(* CODESYS project codesys-syslog-unit-test-history

Project tree, tasks and I/O mapping:
  Device : CODESYS Control Win V3 x64, 3S - Smart Software Solutions GmbH, version 3.5.18.0
    application Application
      libraries: Standard, 3.5.18.0 (System); co♻e - A unittest framework for CODESYS, 1.2.0.0 (www.co5e.org); Code-Syslog Interfaces, * (PowerCore Engineering); CAA File, 3.5.17.0 (CAA Technical Workgroup); CAA Types Extern, 3.5.17.0 (CAA Technical Workgroup); Net Base Services, 3.5.17.0 (3S - Smart Software Solutions GmbH); Element Collections, 3.5.17.0 (3S - Smart Software Solutions GmbH); StringUtils, 3.5.18.0 (System); Code-Syslog, 0.2.0.0 (PowerCore Engineering)
      task MainTask (cyclic, interval t#20ms, priority 1) calls PLC_PRG
      Function Blocks/
        function block UT_SyslogAlarmOnMessageHandler [ST]: T001_TripAlarm, T002_WarnAlarm, T003_RepeatAlarm, T004_RegisterDup
        function block UT_SyslogCaaUdpHandler [ST]: T002_SetupConnection, T003_ProcessQueue
        function block UT_SyslogFileHandler [ST]: AssertEquals_SyslogMsg, CleanUp, T001_FileSetup, T002_ProcessQueue, T003_DiscardWhenFull, T004_FileRemovalRecovery, T999_CleanUp
        function block UT_SyslogLogger [ST]: AssertEquals_SyslogMsg, T001_AppName, T002_Hostname, T003_ProcId, T004_HandlerRegistry, T005_Debug, T006_Info, T007_Notice, T008_Warning, T009_Error, T010_Critical, T011_Alert, T012_Emergency
        function block UT_SyslogRotatingFileHandler [ST]: CleanUp, ls_count, T001_FileSetup, T002_ShouldRollover, T003_Rotate, T004_DoRollover, T005_FullRun, T999_CleanUp
        function block UT_SyslogUdpHandler [ST]: T001_Init, T002_SetupConnection, T003_ProcessQueue
      Functions/
        function block UT_Escape_ParamValue [ST]: T001_Paramaterize
        function block UT_Make_Priority [ST]: T001_Paramaterize
        function block UT_Make_SdParam2 [ST]: T001_Parameterize
        function block UT_Make_SdParam [ST]: T001_Parameterize
        function block UT_RandomEmpherialPort [ST]: T001_Generate
        function block UT_Sanitize_Msg [ST]: T001_Paramaterize
        function block UT_Sanitize_PrintUsAscii [ST]: T001_Paramaterize
        function block UT_Sanitize_SdName [ST]: T001_Paramaterize
        function block UT_StrucDataMsg [ST]: AssertEquals_SyslogMsg, T001_Parameterize
        function block UT_UtcTimestampFromSysTimeDate [ST]: T001_Paramaterize
      Mocks/
        function block Mock_MsgPrependSpace [ST]: AsStructuredData
        function block Mock_StructuredData [ST]: AsStructuredData
        function block Mock_SyslogCaaUdpHandler [ST]: p_QueueBusy, p_uiSendPort, PubProcessQueue, PubSetupConnection, Reset
        function block Mock_SyslogFileHandler [ST]: FileSetup, FlushNow, p_DiscardOldMsgWhenQueueFull, p_FileSize, p_FullFilename, p_mxHandler, p_QueueBusy, PeekQueue, ProcessQueue, ResetQueue
        function block Mock_SyslogHandler [ST]: Dispatch, FB_Init, p_LogSeverity, Reset, Run
        function block Mock_SyslogLogger [ST]: prvTimestamp
        function block Mock_SyslogRotatingFileHandler [ST]: FileSetup, p_FileSize, p_FullFilename, p_hActiveHandle, p_mxHandler, p_QueueBusy, ProcessQueue, PubDoRollover, PubRotate, PubShouldRollover, QueueEmpty, ResetQueue
        function block Mock_SyslogUdpHandler [ST]: AdhockSend, p_QueueBusy, p_uiSendPort, PubInit, PubProcessQueue, PubSetupConnection, Reset
      program PLC_PRG [ST]
      Structs/
        data type ls_data
*)

// Device/Application/Structs/ls_data
TYPE ls_data :
STRUCT
	cFiles : INT;
	szTotalSize : CAA.SIZE;
END_STRUCT
END_TYPE

// Device/Application/PLC_PRG
PROGRAM PLC_PRG
VAR
	utSanitize_PrintUsAscii : UT_Sanitize_PrintUsAscii;
	utSanitize_SdName : UT_Sanitize_SdName;
	utSanitize_Msg : UT_Sanitize_Msg;
	utEscape_ParamValue : UT_Escape_ParamValue;
	utUtcTimestampFromSysTimeDate : UT_UtcTimestampFromSysTimeDate;
	utMake_Priority : UT_Make_Priority;
	utSyslogLogger : UT_SyslogLogger;
	utSyslogFileHandler : UT_SyslogFileHandler;
	utSyslogRotatingFileHandler : UT_SyslogRotatingFileHandler;
	utRandomEmpherialPort : UT_RandomEmpherialPort;
	utSyslogUdpHandler : UT_SyslogUdpHandler;
	utMake_SdParam : UT_Make_SdParam;
	utMake_SdParam2 : UT_Make_SdParam2;
	utStrucDataMsg : UT_StrucDataMsg;
END_VAR

coUnit.RUN_IN_SEQUENCE();

END_PROGRAM

// Device/Application/Functions/UT_Sanitize_PrintUsAscii
FUNCTION_BLOCK UT_Sanitize_PrintUsAscii EXTENDS coUnit.FB_TestSuite
VAR_INPUT
END_VAR
VAR_OUTPUT
END_VAR
VAR
END_VAR

T001_Paramaterize('LegalChars', 
                  'aValidName[don$'t-you_know]',
                  'aValidName[don$'t-you_know]');
T001_Paramaterize('StartWithIllegalChars', 
                  '$n$raValidName[don$'t-you_know]',
                  'aValidName[don$'t-you_know]');
T001_Paramaterize('EndWithIllegalChars', 
                  'aValidName[don$'t-you_know]$de$ad$be$af',
                  'aValidName[don$'t-you_know]');
T001_Paramaterize('IllegalCharsInMiddle', 
                  'aValidName[don$'t-$de$adyou$be$af_know]',
                  'aValidName[don$'t-you_know]');
T001_Paramaterize('AllLegalChars',
                  Syslog.SyslogItfs.gc_sPRINTUSASCII,
                  Syslog.SyslogItfs.gc_sPRINTUSASCII);

METHOD T001_Paramaterize : BOOL
VAR_INPUT
	sTestName : STRING(80);
	sValue : STRING(1000);
	sExpected : STRING(1000);
END_VAR
TEST(sTestName);

Syslog.Sanitize_PrintUsAscii(ADR(sValue));

AssertEquals_BOOL(TRUE, Stu.StrCmpA(ADR(sValue), ADR(sExpected)) = 0, 'sValue does not equal sExpected');

TEST_FINISHED();
END_METHOD

END_FUNCTION_BLOCK

// Device/Application/Functions/UT_Sanitize_SdName
FUNCTION_BLOCK UT_Sanitize_SdName EXTENDS coUnit.FB_TestSuite
VAR_INPUT
END_VAR
VAR_OUTPUT
END_VAR
VAR
END_VAR

T001_Paramaterize('LegalName', 
                  'eventSource',
                  'eventSource');
T001_Paramaterize('StartWithIllegalChars', 
                  '$n$reventSource',
                  'eventSource');
T001_Paramaterize('EndWithIllegalChars', 
                  'eventSource$de$ad$be$af',
                  'eventSource');
T001_Paramaterize('IllegalCharsInMiddle', 
                  'event"]= Source',
                  'eventSource');
T001_Paramaterize('AllLegalChars', 
                  '!#$$%&$'()*+,-./0123456789:;<>?@ABCDEFGHIJKLMNOPQRSTUVWXYZ[\^_`abcdefghijklmnopqrstuvwxyz{|}~',
                  '!#$$%&$'()*+,-./0123456789:;<>?@ABCDEFGHIJKLMNOPQRSTUVWXYZ[\^_`abcdefghijklmnopqrstuvwxyz{|}~');

METHOD T001_Paramaterize : BOOL
VAR_INPUT
	sTestName : STRING(80);
	sValue : STRING(255);
	sExpected : STRING(255);
END_VAR
TEST(sTestName);

Syslog.Sanitize_SdName(ADR(sValue));

AssertEquals_BOOL(TRUE, Stu.StrCmpA(ADR(sValue), ADR(sExpected)) = 0, 'sValue does not equal sExpected');

TEST_FINISHED();
END_METHOD

END_FUNCTION_BLOCK

// Device/Application/Functions/UT_Sanitize_Msg
FUNCTION_BLOCK UT_Sanitize_Msg EXTENDS coUnit.FB_TestSuite
VAR_INPUT
END_VAR
VAR_OUTPUT
END_VAR
VAR
END_VAR

T001_Paramaterize('LegalChars', 
                  '$'su root$' failed for lonvick on /dev/pts/8',
                  '$'su root$' failed for lonvick on /dev/pts/8');
T001_Paramaterize('StartWithIllegalChars', 
                  '$n$r$'su root$' failed for lonvick on /dev/pts/8',
                  '\x0a\x0d$'su root$' failed for lonvick on /dev/pts/8');
T001_Paramaterize('EndWithIllegalChars', 
                  '$'su root$' failed for lonvick on /dev/pts/8$de$ad$be$af$n$r',
                  '$'su root$' failed for lonvick on /dev/pts/8$de$ad$be$af\x0a\x0d');
T001_Paramaterize('IllegalCharsInMiddle', 
                  '$'su root$' failed $de$adfor$be$af$n$r lonvick on /dev/pts/8',
                  '$'su root$' failed $de$adfor$be$af\x0a\x0d lonvick on /dev/pts/8');
T001_Paramaterize('AllLegalChars', 
                  Syslog.SyslogItfs.gc_sPRINTUSASCII,
                  Syslog.SyslogItfs.gc_sPRINTUSASCII);

METHOD T001_Paramaterize : BOOL
VAR_INPUT
	sTestName : STRING(80);
	sValue : STRING(1000);
	sExpected : STRING(1000);
END_VAR
TEST(sTestName);

Syslog.Sanitize_Msg(ADR(sValue), sizeof(sValue));

AssertEquals_BOOL(TRUE, Stu.StrCmpA(ADR(sValue), ADR(sExpected)) = 0, 'sValue does not equal sExpected');

TEST_FINISHED();
END_METHOD

END_FUNCTION_BLOCK

// Device/Application/Functions/UT_Escape_ParamValue
FUNCTION_BLOCK UT_Escape_ParamValue EXTENDS coUnit.FB_TestSuite
VAR_INPUT
END_VAR
VAR_OUTPUT
END_VAR
VAR
END_VAR

T001_Paramaterize('LegalName', 
                  'eventSource',
                  'eventSource');
T001_Paramaterize('StartWithUnescapedChars', 
                  ']"\eventSource',
                  '\]\"\\eventSource');
T001_Paramaterize('EndWithUnescapedChars', 
                  'eventSource]"\',
                  'eventSource\]\"\\');
T001_Paramaterize('UnescapedCharsInMiddle', 
                  'event"]\Source',
                  'event\"\]\\Source');
T001_Paramaterize('MixOfEscapedAndUnescaped', 
                  'event\"\\So\ur]ce',
                  'event\"\\So\\ur\]ce');
T001_Paramaterize('AllLegalChars', 
                  '!#$$%&$'()*+,-./0123456789:;<=>?@ABCDEFGHIJKLMNOPQRSTUVWXYZ[^_`abcdefghijklmnopqrstuvwxyz{|}~',
                  '!#$$%&$'()*+,-./0123456789:;<=>?@ABCDEFGHIJKLMNOPQRSTUVWXYZ[^_`abcdefghijklmnopqrstuvwxyz{|}~');

METHOD T001_Paramaterize : BOOL
VAR_INPUT
	sTestName : STRING(80);
	sValue : STRING(255);
	sExpected : STRING(255);
END_VAR
TEST(sTestName);

Syslog.Escape_ParamValue(ADR(sValue), sizeof(sValue));

AssertEquals_BOOL(TRUE, Stu.StrCmpA(ADR(sValue), ADR(sExpected)) = 0, 'sValue does not equal sExpected');

TEST_FINISHED();
END_METHOD

END_FUNCTION_BLOCK

// Device/Application/Functions/UT_UtcTimestampFromSysTimeDate
FUNCTION_BLOCK UT_UtcTimestampFromSysTimeDate EXTENDS coUnit.FB_TestSuite
VAR_INPUT
END_VAR
VAR_OUTPUT
END_VAR
VAR
	rtsNull : Syslog.SysTimeRtc.SYSTIMEDATE;
	// 2003-10-11T22:14:15.003Z
	rtsRfcExample3 : Syslog.SysTimeRtc.SYSTIMEDATE := (wYear:=2003, wMonth:=10, wDay:=11, wHour:=22, wMinute:=14, wSecond:=15, wMilliseconds:=3);
	rtsSingleDigits : Syslog.SysTimeRtc.SYSTIMEDATE := (wYear:=2003, wMonth:=1, wDay:=1, wHour:=2, wMinute:=4, wSecond:=5, wMilliseconds:=3);
END_VAR

T001_Paramaterize('NullDate', 
                  rtsNull,
                  '0000-00-00T00:00:00.000Z');
T001_Paramaterize('RfcExample3', 
                  rtsRfcExample3,
                  '2003-10-11T22:14:15.003Z');
T001_Paramaterize('SingleDigits', 
                  rtsSingleDigits,
                  '2003-01-01T02:04:05.003Z');

METHOD T001_Paramaterize : BOOL
VAR_INPUT
	sTestName : STRING(80);
	rts : Syslog.SysTimeRtc.SYSTIMEDATE;
	sExpected : STRING(255);
END_VAR
VAR
	sTimestamp : Syslog.SyslogItfs.TIMESTAMP;
END_VAR
TEST(sTestName);

sTimestamp := Syslog.UtcTimestampFromSystimeDate(rts);

AssertEquals_STRING(sExpected, sTimestamp, 'Timestamps do not match');

TEST_FINISHED();
END_METHOD

END_FUNCTION_BLOCK

// Device/Application/Functions/UT_Make_Priority
FUNCTION_BLOCK UT_Make_Priority EXTENDS coUnit.FB_TestSuite
VAR_INPUT
END_VAR
VAR_OUTPUT
END_VAR
VAR
END_VAR

T001_Paramaterize('Kern emerg', Syslog.SyslogItfs.SyslogSeverity.EMERGENCY, Syslog.SyslogItfs.SyslogFacility.KERN, '<0>');
T001_Paramaterize('user alert', Syslog.SyslogItfs.SyslogSeverity.ALERT, Syslog.SyslogItfs.SyslogFacility.USER, '<9>');
T001_Paramaterize('local notice', Syslog.SyslogItfs.SyslogSeverity.NOTICE, Syslog.SyslogItfs.SyslogFacility.LOCAL4, '<165>');

METHOD T001_Paramaterize : BOOL
VAR_INPUT
	sTestName : STRING(255);
	sev : Syslog.SyslogItfs.SyslogSeverity;
	fac : Syslog.SyslogItfs.SyslogFacility;
	sExpected : STRING(10);
END_VAR
VAR
	pri : Syslog.SyslogItfs.PRI;
END_VAR
TEST(sTestName);

pri := Syslog.Make_Priority(sev, fac);

AssertEquals_STRING(pri, sExpected, 'PRI does not equal sExpected');

TEST_FINISHED();
END_METHOD

END_FUNCTION_BLOCK

// Device/Application/Function Blocks/UT_SyslogLogger
FUNCTION_BLOCK UT_SyslogLogger EXTENDS coUnit.FB_TestSuite
VAR_INPUT
END_VAR
VAR_OUTPUT
END_VAR
VAR
	handler : Mock_SyslogHandler(severity:=SyslogItfs.SyslogSeverity.DEBUG);
	itfHandler : SyslogItfs.ISyslogHandler := handler;
	// local4 = 20 to make manual pri easier to calculate. 20*8 = 160
	logger : Mock_SyslogLogger(hostname:='codesyslog.example.com', appName:='UnitTest', procId:='PLC_PRG', facility:=SyslogItfs.SyslogFacility.LOCAL4, handler:=itfHandler);
END_VAR

T001_AppName('T001_AppName:EmptyAppName', '', SyslogItfs.gc_sNILVALUE);
T001_AppName('T001_AppName:InvalidCharsRemoved', '$nUnit Test', 'UnitTest');

T002_Hostname('T002_Hostname:EmptyHostname', '$n $r', SyslogItfs.gc_sNILVALUE);
T002_Hostname('T002_Hostname:InvalidCharsRemoved', 'invalid hostname', 'invalidhostname');
T002_Hostname('T002_Hostname:IPAddress', '192.168.0.1', '192.168.0.1');
T002_Hostname('T002_Hostname:FQDN', 'codesyslog.example.com', 'codesyslog.example.com');

T003_ProcId('T003_ProcId:EmptyProcId', '', SyslogItfs.gc_sNILVALUE);
T003_ProcId('T003_ProcId:InvalidCharsRemoved', '$de$ad$be$efPLC_PRG', 'PLC_PRG');

T004_HandlerRegistry();
T005_Debug();
T006_Info();
T007_Notice();
T008_Warning();
T009_Error();
T010_Critical();
T011_Alert();
T012_Emergency();

METHOD AssertEquals_SyslogMsg
VAR_INPUT
	actual : POINTER TO SyslogItfs.SYSLOG_MSG;
	expected : POINTER TO SyslogItfs.SYSLOG_MSG;
END_VAR
VAR
	ix : UINT;
	pa : POINTER TO ARRAY [0..SyslogItfs.gc_szSyslogMsg-1] OF BYTE := actual;
	pe : POINTER TO ARRAY [0..SyslogItfs.gc_szSyslogMsg-1] OF BYTE := expected;
	xDifferent : BOOL;
END_VAR
FOR ix := 0 TO SyslogItfs.gc_szSyslogMsg-1 BY 1 DO
	IF pa^[ix] <> 0 AND pe^[ix] <> 0 THEN
		IF pa^[ix] <> pe^[ix] THEN
			xDifferent := TRUE;
			EXIT;
		END_IF
	ELSIF pa^[ix] = 0 AND pe^[ix] = 0 THEN
		EXIT;
	ELSE
		xDifferent := TRUE;
		EXIT;
	END_IF
END_FOR

AssertFalse(xDifferent, concat('SYSLOG_MSG found to differ at character: ', UINT_TO_STRING(ix)));
END_METHOD

METHOD T001_AppName
VAR_INPUT
	sTestName : STRING(255);
	sAppName : SyslogItfs.APP_NAME;
	sExpected : SyslogItfs.APP_NAME;
END_VAR
VAR
	sResult : SyslogItfs.APP_NAME;
END_VAR
IF TEST_ORDERED(sTestName) THEN

	logger.SetAppName(sAppName);
	sResult := logger.GetAppName();
	
	AssertEquals_STRING(sExpected, sResult, 'Unexpected AppName');
	
	TEST_FINISHED();
END_IF
END_METHOD

METHOD T002_Hostname
VAR_INPUT
	sTestName : STRING(255);
	sValue : SyslogItfs.HOSTNAME;
	sExpected : SyslogItfs.HOSTNAME;
END_VAR
VAR
	sResult : SyslogItfs.HOSTNAME;
END_VAR
IF TEST_ORDERED(sTestName) THEN

	logger.SetHostname(sValue);
	sResult := logger.GetHostname();
	
	AssertEquals_STRING(sExpected, sResult, 'Unexpected Hostname');
	
	TEST_FINISHED();
END_IF
END_METHOD

METHOD T003_ProcId
VAR_INPUT
	sTestName : STRING(255);
	sValue : SyslogItfs.PROC_ID;
	sExpected : SyslogItfs.PROC_ID;
END_VAR
VAR
	sResult : SyslogItfs.PROC_ID;
END_VAR
IF TEST_ORDERED(sTestName) THEN

	logger.SetProcId(sValue);
	sResult := logger.GetProcId();
	
	AssertEquals_STRING(sExpected, sResult, 'Unexpected Proc ID');
	
	TEST_FINISHED();
END_IF
END_METHOD

METHOD T004_HandlerRegistry
VAR_INPUT
END_VAR
VAR
	xResult : BOOL;
END_VAR
IF TEST_ORDERED('T004_HandlerRegistry') THEN

	xResult := logger.RegisterHandler(itfHandler);
	AssertFalse(xResult, 'Handle registered twice!');
	
	xResult := logger.UnregisterHandler(itfHandler);
	AssertTrue(xResult, 'Handle failed to unregistered');
	
	xResult := logger.RegisterHandler(itfHandler);
	AssertTrue(xResult, 'Handle failed to registered');
	
	TEST_FINISHED();
END_IF
END_METHOD

METHOD T005_Debug
VAR_INPUT
END_VAR
VAR
	expected : SyslogItfs.SYSLOG_MSG;
END_VAR
IF TEST_ORDERED('T005_Debug') THEN

	logger.Debug('DEBUG', 'lorum ipsum');
	expected := '<167>1 2021-11-22T23:40:05.003Z codesyslog.example.com UnitTest PLC_PRG DEBUG lorum ipsum';
	AssertEquals_SyslogMsg(ADR(handler.lastMessage), ADR(expected));
	
	handler.Reset();
	handler.p_LogSeverity := SyslogItfs.SyslogSeverity.INFORMATION;
	
	logger.Debug('DEBUG', 'lorum ipsum');
	expected := '';
	AssertEquals_SyslogMsg(ADR(handler.lastMessage), ADR(expected));
	
	
	TEST_FINISHED();
END_IF
END_METHOD

METHOD T006_Info
VAR_INPUT
END_VAR
VAR
	expected : SyslogItfs.SYSLOG_MSG;
END_VAR
IF TEST_ORDERED('T006_Info') THEN

	logger.Information('INFO', 'lorum ipsum');
	expected := '<166>1 2021-11-22T23:40:05.003Z codesyslog.example.com UnitTest PLC_PRG INFO lorum ipsum';
	AssertEquals_SyslogMsg(ADR(handler.lastMessage), ADR(expected));
	
	handler.Reset();
	handler.p_LogSeverity := SyslogItfs.SyslogSeverity.NOTICE;
	
	logger.Information('INFO', 'lorum ipsum');
	expected := '';
	AssertEquals_SyslogMsg(ADR(handler.lastMessage), ADR(expected));
	
	
	TEST_FINISHED();
END_IF
END_METHOD

METHOD T007_Notice
VAR_INPUT
END_VAR
VAR
	expected : SyslogItfs.SYSLOG_MSG;
END_VAR
IF TEST_ORDERED('T007_Notice') THEN

	logger.Notice('NOTICE', 'lorum ipsum');
	expected := '<165>1 2021-11-22T23:40:05.003Z codesyslog.example.com UnitTest PLC_PRG NOTICE lorum ipsum';
	AssertEquals_SyslogMsg(ADR(handler.lastMessage), ADR(expected));
	
	handler.Reset();
	handler.p_LogSeverity := SyslogItfs.SyslogSeverity.WARNING;
	
	logger.Notice('NOTICE', 'lorum ipsum');
	expected := '';
	AssertEquals_SyslogMsg(ADR(handler.lastMessage), ADR(expected));
	
	
	TEST_FINISHED();
END_IF
END_METHOD

METHOD T008_Warning
VAR_INPUT
END_VAR
VAR
	expected : SyslogItfs.SYSLOG_MSG;
END_VAR
IF TEST_ORDERED('T008_Warning') THEN

	logger.Warning('WARN', 'lorum ipsum');
	expected := '<164>1 2021-11-22T23:40:05.003Z codesyslog.example.com UnitTest PLC_PRG WARN lorum ipsum';
	AssertEquals_SyslogMsg(ADR(handler.lastMessage), ADR(expected));
	
	handler.Reset();
	handler.p_LogSeverity := SyslogItfs.SyslogSeverity.ERROR;
	
	logger.Warning('WARN', 'lorum ipsum');
	expected := '';
	AssertEquals_SyslogMsg(ADR(handler.lastMessage), ADR(expected));
	
	
	TEST_FINISHED();
END_IF
END_METHOD

METHOD T009_Error
VAR_INPUT
END_VAR
VAR
	expected : SyslogItfs.SYSLOG_MSG;
END_VAR
IF TEST_ORDERED('T009_Error') THEN

	logger.Error('ERROR', 'lorum ipsum');
	expected := '<163>1 2021-11-22T23:40:05.003Z codesyslog.example.com UnitTest PLC_PRG ERROR lorum ipsum';
	AssertEquals_SyslogMsg(ADR(handler.lastMessage), ADR(expected));
	
	handler.Reset();
	handler.p_LogSeverity := SyslogItfs.SyslogSeverity.CRITICAL;
	
	logger.Error('ERROR', 'lorum ipsum');
	expected := '';
	AssertEquals_SyslogMsg(ADR(handler.lastMessage), ADR(expected));
	
	
	TEST_FINISHED();
END_IF
END_METHOD

METHOD T010_Critical
VAR_INPUT
END_VAR
VAR
	expected : SyslogItfs.SYSLOG_MSG;
END_VAR
IF TEST_ORDERED('T010_Critical') THEN

	logger.Critical('CRITICAL', 'lorum ipsum');
	expected := '<162>1 2021-11-22T23:40:05.003Z codesyslog.example.com UnitTest PLC_PRG CRITICAL lorum ipsum';
	AssertEquals_SyslogMsg(ADR(handler.lastMessage), ADR(expected));
	
	handler.Reset();
	handler.p_LogSeverity := SyslogItfs.SyslogSeverity.ALERT;
	
	logger.Critical('CRITICAL', 'lorum ipsum');
	expected := '';
	AssertEquals_SyslogMsg(ADR(handler.lastMessage), ADR(expected));
	
	
	TEST_FINISHED();
END_IF
END_METHOD

METHOD T011_Alert
VAR_INPUT
END_VAR
VAR
	expected : SyslogItfs.SYSLOG_MSG;
END_VAR
IF TEST_ORDERED('T011_Alert') THEN

	logger.Alert('ALERT', 'lorum ipsum');
	expected := '<161>1 2021-11-22T23:40:05.003Z codesyslog.example.com UnitTest PLC_PRG ALERT lorum ipsum';
	AssertEquals_SyslogMsg(ADR(handler.lastMessage), ADR(expected));
	
	handler.Reset();
	handler.p_LogSeverity := SyslogItfs.SyslogSeverity.EMERGENCY;
	
	logger.Alert('ALERT', 'lorum ipsum');
	expected := '';
	AssertEquals_SyslogMsg(ADR(handler.lastMessage), ADR(expected));
	
	
	TEST_FINISHED();
	END_IF
END_METHOD

METHOD T012_Emergency
VAR_INPUT
END_VAR
VAR
	expected : SyslogItfs.SYSLOG_MSG;
END_VAR
IF TEST_ORDERED('T012_Emergency') THEN

	logger.Emergency('EMERGENCY', 'lorum ipsum');
	expected := '<160>1 2021-11-22T23:40:05.003Z codesyslog.example.com UnitTest PLC_PRG EMERGENCY lorum ipsum';
	AssertEquals_SyslogMsg(ADR(handler.lastMessage), ADR(expected));
	
	handler.Reset();
	handler.p_LogSeverity := SyslogItfs.SyslogSeverity.DEBUG;
	
	logger.Emergency('EMERGENCY', 'lorum ipsum debug');
	expected := '<160>1 2021-11-22T23:40:05.003Z codesyslog.example.com UnitTest PLC_PRG EMERGENCY lorum ipsum debug';
	AssertEquals_SyslogMsg(ADR(handler.lastMessage), ADR(expected));
	
	
	TEST_FINISHED();
END_IF
END_METHOD

END_FUNCTION_BLOCK

// Device/Application/Mocks/Mock_SyslogHandler
/// This syslog handler doesn't only stores the last value dispatched
FUNCTION_BLOCK Mock_SyslogHandler IMPLEMENTS SyslogItfs.ISyslogHandler
VAR_INPUT
END_VAR
VAR_OUTPUT
	lastMessage : SyslogItfs.SYSLOG_MSG;
END_VAR
VAR
	_severity : SyslogItfs.SyslogSeverity;
END_VAR

METHOD Dispatch : BOOL
VAR_INPUT
	syslogMsg	: SyslogItfs.SYSLOG_MSG;
END_VAR
THIS^.lastMessage := syslogMsg;
END_METHOD

//FB_Init is always available implicitly and it is used primarily for initialization.
//The return value is not evaluated. For a specific influence, you can also declare the
//methods explicitly and provide additional code there with the standard initialization
//code. You can evaluate the return value.
METHOD FB_Init: BOOL
VAR_INPUT
    bInitRetains: BOOL; // TRUE: the retain variables are initialized (reset warm / reset cold)
    bInCopyCode: BOOL;  // TRUE: the instance will be copied to the copy code afterward (online change)   
	severity : SyslogItfs.SyslogSeverity;
END_VAR
THIS^._severity := severity;
END_METHOD

{attribute 'monitoring' := 'call'}
PROPERTY p_LogSeverity : SyslogItfs.SyslogSeverity
GET
p_LogSeverity := this^._severity;
END_GET
SET
this^._severity := p_LogSeverity;
END_SET
END_PROPERTY

METHOD Reset : BOOL
VAR_INPUT
END_VAR
lastMessage := '';
END_METHOD

(* Run the handler base code*)
METHOD Run : BOOL
END_METHOD

END_FUNCTION_BLOCK

// Device/Application/Mocks/Mock_SyslogLogger
FUNCTION_BLOCK Mock_SyslogLogger EXTENDS Syslog.SyslogLogger
VAR_INPUT
END_VAR
VAR_OUTPUT
END_VAR
VAR
END_VAR

/// prvTimestamp exists so we can override the timestamp for testing
METHOD PROTECTED prvTimestamp : Syslog.SyslogItfs.TIMESTAMP
VAR_INPUT
END_VAR
VAR
	// 2021-11-22T23:40:05.003Z
	rts : Syslog.SysTimeRtc.SYSTIMEDATE := (wYear:=2021, wMonth:=11, wDay:=22, wHour:=23, wMinute:=40, wSecond:=5, wMilliseconds:=3);
END_VAR
prvTimestamp := Syslog.UtcTimestampFromSystimeDate(rts);
END_METHOD

END_FUNCTION_BLOCK

// Device/Application/Function Blocks/UT_SyslogFileHandler
FUNCTION_BLOCK UT_SyslogFileHandler EXTENDS coUnit.FB_TestSuite
VAR_INPUT
END_VAR
VAR_OUTPUT
END_VAR
VAR
	handler : Mock_SyslogFileHandler;
END_VAR

T001_FileSetup();
T002_ProcessQueue();
T003_DiscardWhenFull();
T004_FileRemovalRecovery();


// Final cleanup
T999_CleanUp();

METHOD AssertEquals_SyslogMsg
VAR_INPUT
	actual : POINTER TO SyslogItfs.SYSLOG_MSG;
	expected : POINTER TO SyslogItfs.SYSLOG_MSG;
END_VAR
VAR
	ix : UINT;
	pa : POINTER TO ARRAY [0..SyslogItfs.gc_szSyslogMsg-1] OF BYTE := actual;
	pe : POINTER TO ARRAY [0..SyslogItfs.gc_szSyslogMsg-1] OF BYTE := expected;
	xDifferent : BOOL;
END_VAR
FOR ix := 0 TO SyslogItfs.gc_szSyslogMsg-1 BY 1 DO
	IF pa^[ix] <> 0 AND pe^[ix] <> 0 THEN
		IF pa^[ix] <> pe^[ix] THEN
			xDifferent := TRUE;
			EXIT;
		END_IF
	ELSIF pa^[ix] = 0 AND pe^[ix] = 0 THEN
		EXIT;
	ELSE
		xDifferent := TRUE;
		EXIT;
	END_IF
END_FOR

AssertFalse(xDifferent, concat('SYSLOG_MSG found to differ at character: ', UINT_TO_STRING(ix)));
END_METHOD

METHOD CleanUp : BOOL;
VAR_INPUT
END_VAR
VAR_INST
	rmdir : FILE.DirRemove;
END_VAR
rmdir(xExecute:=TRUE, sDirName:='csyslog/', xRecursive:=TRUE);
IF rmdir.xDone OR rmdir.xError THEN
	CleanUp := TRUE;
	rmdir(xExecute:=FALSE);
END_IF
END_METHOD

METHOD T001_FileSetup
VAR_INPUT
END_VAR
VAR_INST
	tmr : TON := (PT:=T#5S);
	mxFileSetup : UINT;
	getSize : FILE.GetSize;
END_VAR
IF TEST_ORDERED('T001_FileSetup') THEN
	tmr(IN:=TRUE);
	CASE mxFileSetup OF
		0: // Run file setup
			IF handler.FileSetup() OR tmr.Q OR handler.xError THEN
				mxFileSetup := 10;
			END_IF
		10: // Simple Asserts
			AssertFalse(handler.xError, 'Error after file setup');
			AssertFalse(tmr.Q, 'FileSetup timed out');
			mxFileSetup := 20;
		20: // check filesystem
			getSize(xExecute:=TRUE, sFileName:=handler.p_FullFilename);
			IF getSize.xDone OR getSize.xError THEN
				AssertFalse(getSize.xError, concat('An error occured getting file size. Error: ', TO_STRING(getSize.eError)));
				AssertFalse(getSize.xError, concat('Error on file: ', TO_STRING(handler.p_FullFilename)));
				getSize(xExecute:=FALSE);
				mxFileSetup := 30;
			END_IF
		ELSE
			TEST_FINISHED();
	END_CASE
	
	
END_IF
END_METHOD

METHOD T002_ProcessQueue
VAR_INPUT
END_VAR
VAR_INST
	mxT : UINT;
	tmr : TON := (PT:=T#5S);
	fileSize : FILE.GetSize;
END_VAR
IF TEST_ORDERED('T002_ProcessQueue') THEN
	CASE mxT OF
		0: // setup
			handler.Dispatch('hello, world');
			handler.Dispatch('<167>1 2021-11-22T23:40:05.003Z codesyslog.example.com UnitTest PLC_PRG DEBUG lorum ipsum');
			mxT := 10;
		10: // run queue process for 5 seconds
			tmr(IN:=TRUE);
			handler.ProcessQueue();
			IF tmr.Q OR NOT handler.p_QueueBusy THEN
				AssertFalse(tmr.Q, 'ProcessQueue timeout');
				tmr(IN:=FALSE);
				mxT := 20;
			END_IF
		20: // get fileSize
			fileSize(xExecute:=TRUE, sFileName:=handler.p_FullFilename);
			IF fileSize.xDone OR fileSize.xError THEN
				AssertFalse(fileSize.xError, 'Error getting file size');
				AssertEquals_UDINT(handler.p_FileSize, __UXINT_TO_UDINT(fileSize.szSize), 'calculated file size and actual file size do not match');
				fileSize(xExecute:=FALSE); 
				mxT := 30;
			END_IF
		30: // other asserts
			AssertFalse(handler.xError, 'Error during queue processing');
			mxT := 40;
		ELSE
			TEST_FINISHED();
	END_CASE
END_IF
END_METHOD

METHOD T003_DiscardWhenFull
VAR_INPUT
END_VAR
VAR_INST
	mxT : UINT;
	ix : UINT;
	sHead : SyslogItfs.SYSLOG_MSG;
	sExpected : STRING(10) := '21';
END_VAR
IF TEST_ORDERED('T003_DiscardWhenFull') THEN
	CASE mxT OF
		0: // init
			handler.p_DiscardOldMsgWhenQueueFull := TRUE;
			FOR ix := 0 TO 1020 BY 1 DO
				handler.Dispatch(UINT_TO_STRING(ix));
			END_FOR
			mxT := 10;
		10: // check for overrun
			sHead := handler.PeekQueue();
			AssertEquals_STRING(sExpected, sHead, 'Queue head unexpected value');
			handler.ResetQueue();
			handler.p_DiscardOldMsgWhenQueueFull := FALSE;
			mxT := 20;
		ELSE
			TEST_FINISHED();
	END_CASE
END_IF
END_METHOD

METHOD T004_FileRemovalRecovery
VAR_INPUT
END_VAR
VAR_INST
	mxT : UINT;
	tmr : TON := (PT:=T#10s);
END_VAR
IF TEST_ORDERED('T004_FileRemovalRecovery') THEN
	CASE mxT OF
		0: // setup
			// run until in process queue
			handler.Run();
			IF handler.p_mxHandler = 10 THEN
				// remove directory and file
				IF CleanUp() THEN
					mxT := 10;
				END_IF
			END_IF
		10: // dispatch a message
			handler.Dispatch('write to missing file');
			mxT := 20;
		20: // run until back in init mode
			handler.Run();
			tmr(IN:=TRUE);
			IF handler.p_mxHandler = 0 OR tmr.Q THEN
				AssertFalse(tmr.Q, 'handler.Run() until timeout mxT=20');
				AssertFalse(handler.xError, 'handler.xError mxT=20');
				tmr(IN:=FALSE);
				mxT := 30;
			END_IF
		30: // run until idle (should never have stopped being busy during reset)
			handler.Run();
			tmr(IN:=TRUE);
			IF (handler.p_mxHandler = 10 AND NOT handler.p_QueueBusy) OR tmr.Q THEN
				AssertFalse(tmr.Q, 'handler.Run() until timeout mxT=30');
				AssertFalse(handler.xError, 'handler.xError mxT=30');
				mxT := 40;
			END_IF
		ELSE
			TEST_FINISHED();
	END_CASE
END_IF
END_METHOD

METHOD T999_CleanUp
VAR_INPUT
END_VAR
IF TEST_ORDERED('T999_CleanUp') THEN
	IF CleanUp() THEN
		AssertTrue(TRUE, 'cleaned up');
		TEST_FINISHED();
	END_IF
END_IF
END_METHOD

END_FUNCTION_BLOCK

// Device/Application/Mocks/Mock_SyslogFileHandler
FUNCTION_BLOCK Mock_SyslogFileHandler EXTENDS Syslog.SyslogFileHandler
VAR_INPUT
END_VAR
VAR_OUTPUT
END_VAR
VAR
END_VAR

METHOD FileSetup : BOOL
VAR_INPUT
END_VAR
FileSetup := prvFileSetup();
END_METHOD

METHOD FlushNow : BOOL
VAR_INPUT
END_VAR
FlushNow := THIS^.prvFlush();
END_METHOD

PROPERTY p_DiscardOldMsgWhenQueueFull : BOOL
GET
p_DiscardOldMsgWhenQueueFull := THIS^.xDiscardOldMsgWhenQueueFull;
END_GET
SET
THIS^.xDiscardOldMsgWhenQueueFull := p_DiscardOldMsgWhenQueueFull;
END_SET
END_PROPERTY

{attribute 'monitoring' := 'call'}
PROPERTY p_FileSize : UDINT
GET
p_FileSize := THIS^.szFilesize;
END_GET
END_PROPERTY

{attribute 'monitoring' := 'call'}
PROPERTY p_FullFilename : CAA.FILENAME
GET
p_FullFilename := THIS^.sFullFilename;
END_GET
END_PROPERTY

PROPERTY p_mxHandler : UINT
GET
p_mxHandler := mxHandler;
END_GET
END_PROPERTY

PROPERTY p_QueueBusy : BOOL
GET
p_QueueBusy := xQueueBusy;
END_GET
END_PROPERTY

METHOD PeekQueue : SyslogItfs.SYSLOG_MSG
VAR_INPUT
END_VAR
queue.Peek(itfElement => THIS^.itfElement);
IF __QUERYINTERFACE(itfElement, itfSyslogMsgElement) THEN
	PeekQueue := itfSyslogMsgElement.SyslogMsgValue;
END_IF
END_METHOD

METHOD ProcessQueue : BOOL
VAR_INPUT
END_VAR
ProcessQueue := prvProcessQueue();
END_METHOD

METHOD ResetQueue : BOOL
VAR_INPUT
END_VAR
this^.queue.RemoveAllElements();
END_METHOD

END_FUNCTION_BLOCK

// Device/Application/Function Blocks/UT_SyslogRotatingFileHandler
FUNCTION_BLOCK UT_SyslogRotatingFileHandler EXTENDS coUnit.FB_TestSuite
VAR_INPUT
END_VAR
VAR_OUTPUT
END_VAR
VAR
	handler : Mock_SyslogRotatingFileHandler := (szMaxFilesize:=1024, uiBackupCount:=3);
END_VAR

T001_FileSetup();
T002_ShouldRollover();
T003_Rotate();
T004_DoRollover();
T005_FullRun();

//T999_CleanUp();

METHOD CleanUp : BOOL;
VAR_INPUT
END_VAR
VAR_INST
	rmdir : FILE.DirRemove;
END_VAR
rmdir(xExecute:=TRUE, sDirName:='csyslog/', xRecursive:=TRUE);
IF rmdir.xDone OR rmdir.xError THEN
	CleanUp := TRUE;
	rmdir(xExecute:=FALSE);
END_IF
END_METHOD

METHOD ls_count : ls_data
VAR_INPUT
END_VAR
VAR_INST
	mxT : UINT;
	hDir : CAA.HANDLE;
	dopen : FILE.DirOpen;
	dclose : FILE.DirClose;
	dls : FILE.DirList;
	lsd : ls_data;
END_VAR
ls_count.cFiles := -1;
CASE mxT OF
	0: // open dir
		lsd.cFiles := 0;
		lsd.szTotalSize := 0;
		dopen(xExecute:=TRUE, sDirName:='csyslog/');
		IF dopen.xDone OR dopen.xError THEN
			AssertFalse(dopen.xError, 'Error opening dir');
			hDir := dopen.hDir;
			dopen(xExecute:=FALSE);
			mxT := 20;
		END_IF
	20: // list and count files
		dls(xExecute:=TRUE, hDir:=hDir);
		IF dls.xDone OR dls.xError THEN
			IF NOT dls.xError THEN
				IF dls.deDirEntry.sEntry <> '.' AND dls.deDirEntry.sEntry <> '..' THEN
					lsd.cFiles := lsd.cFiles + 1;
					lsd.szTotalSize := lsd.szTotalSize + dls.deDirEntry.szSize;
				END_IF
			ELSE
				mxT := 30;
			END_IF
			dls(xExecute:=FALSE);
		END_IF
	30: // close dir
		dclose(xExecute:=TRUE, hDir:=hDir);
		IF dclose.xDone OR dclose.xError THEN
			hDir := CAA.gc_hINVALID;
			dclose(xExecute:=FALSE);
			mxT := 0;
			ls_count := lsd;
		END_IF
END_CASE
END_METHOD

METHOD T001_FileSetup
VAR_INPUT
END_VAR
VAR_INST
	tmr : TON := (PT:=T#5S);
	mxFileSetup : UINT;
	getSize : FILE.GetSize;
END_VAR
IF TEST_ORDERED('T001_FileSetup') THEN
	tmr(IN:=TRUE);
	CASE mxFileSetup OF
		0: // Run file setup
			IF handler.FileSetup() OR tmr.Q OR handler.xError THEN
				mxFileSetup := 10;
			END_IF
		10: // Simple Asserts
			AssertFalse(handler.xError, 'Error after file setup');
			AssertFalse(tmr.Q, 'FileSetup timed out');
			mxFileSetup := 20;
		20: // check filesystem
			getSize(xExecute:=TRUE, sFileName:=handler.p_FullFilename);
			IF getSize.xDone OR getSize.xError THEN
				AssertFalse(getSize.xError, concat('An error occured getting file size. Error: ', TO_STRING(getSize.eError)));
				AssertFalse(getSize.xError, concat('Error on file: ', TO_STRING(handler.p_FullFilename)));
				getSize(xExecute:=FALSE);
				mxFileSetup := 30;
			END_IF
		ELSE
			TEST_FINISHED();
	END_CASE
	
	
END_IF
END_METHOD

METHOD T002_ShouldRollover
VAR_INPUT
END_VAR
VAR
	xResult : BOOL;
END_VAR
IF TEST_ORDERED('T002_ShouldRollover') THEN
	handler.p_FileSize := UDINT#1024;
	xResult := handler.PubShouldRollover();
	AssertFalse(xResult, 'completely full, but no message in queue');
	
	// add a message
	handler.Dispatch('hello, world'); // 12 bytes + $n = 13 bytes
	
	handler.p_FileSize := UDINT#1024 - 13;
	xResult := handler.PubShouldRollover();
	AssertFalse(xResult, 'should completely fill, but not rollover yet');
	
	handler.p_FileSize := UDINT#1024 - 12;
	xResult := handler.PubShouldRollover();
	AssertTrue(xResult, 'should rollover');
	
	handler.p_FileSize := 0;
	xResult := handler.PubShouldRollover();
	AssertFalse(xResult, 'should not rollover at 0');
	
	// reset handler
	handler.p_FileSize := 0;
	handler.ResetQueue();
	
	TEST_FINISHED();
END_IF
END_METHOD

METHOD T003_Rotate
VAR_INPUT
END_VAR
VAR_INST
	mxT : UINT;
	hHandle : CAA.HANDLE;
	sDest : CAA.FILENAME;
	fileSize : FILE.GetSize;
END_VAR
IF TEST_ORDERED('T003_Rotate') THEN
	CASE mxT OF
		0: // init
			hHandle := handler.p_hActiveHandle;
			sDest := concat(handler.p_FullFilename, '.1');
			mxT := 10;
		10: // rotate
			IF handler.PubRotate(handler.p_FullFilename, sDest) THEN
				mxT := 20;
			END_IF
		20: // get size
			fileSize(xExecute:=TRUE, sFileName:=sDest);
			IF fileSize.xError OR fileSize.xDone THEN
				AssertFalse(filesize.xError, 'sDest file should exist, but does not');
				fileSize(xExecute:=FALSE);
				mxT := 30;
			END_IF
		30: // check handle
			// we aren't guarenteed a new handle pointer value even if we close and open a file.
			//AssertFalse(CAA.HANDLE_TO_DWORD(hHandle) = CAA.HANDLE_TO_DWORD(handler.p_hActiveHandle), 'should have a new file handle');
			AssertFalse(CAA.gc_hINVALID = CAA.HANDLE_TO_DWORD(handler.p_hActiveHandle), 'should be a valid handle');
			mxT := 40;
		ELSE
			TEST_FINISHED();
	END_CASE
END_IF
END_METHOD

METHOD T004_DoRollover
VAR_INPUT
END_VAR
VAR_INST
	mxT: UINT;
	lsd : ls_data;
END_VAR
IF TEST_ORDERED('T004_DoRollover') THEN
	CASE mxT OF
		0: // Do the roll over
			IF handler.PubDoRollover() THEN
				mxT := 10;
			END_IF
		10: // count files
			lsd := ls_count();
			IF lsd.cFiles >= 0 THEN
				mxT := 40;
			END_IF
		40: // asserts
			AssertEquals_INT(3, lsd.cFiles, 'unexpected number of files after rollover');
			mxT := 50;
		ELSE
			TEST_FINISHED();
	END_CASE
END_IF
END_METHOD

METHOD T005_FullRun
VAR_INPUT
END_VAR
VAR_INST
	mxT : UINT;
	ix : UINT;
	msg : SyslogItfs.SYSLOG_MSG := ' ';
	sRow : STRING(1) := '1';
	tickStart : CAA.TICK;
	tickEnd : CAA.TICK;
	tickDiff : CAA.TICK;
	lsd : ls_data;
	szExpected : CAA.SIZE := 3328; // 13 * 256
END_VAR
IF TEST_ORDERED('T005_FullRun') THEN
	CASE mxT OF 
		0: // fill queue with enough data for 4 DoRollover
			FOR ix := 0 TO 12 BY 1 DO
				sRow := UINT_TO_STRING(ix);
				Stu.StrPadLeftA(UINT_TO_BYTE(ix) + SyslogItfs.gc_byZERO_DIGIT, ADR(sRow), ADR(msg), 255);
				handler.Dispatch(msg);
			END_FOR
			mxT := 10;
			tickStart := FILE.TICKS.GetTick(TRUE);
		10: // run until done
			handler.Run();
			IF handler.QueueEmpty() AND NOT handler.p_QueueBusy THEN
				handler.p_FlushNow := TRUE;
				mxT := 15;
				tickEnd := FILE.TICKS.GetTick(TRUE);
				tickDiff := tickEnd - tickStart;
			END_IF
		15: // run until flush done
			handler.Run();
			IF NOT handler.p_FlushNow THEN
				mxT := 20;
			END_IF
		20: // number of files
			lsd := ls_count();
			IF lsd.cFiles >= 0 THEN
				mxT := 30;
			END_IF
		30: // asserts
			AssertEquals_INT(4, lsd.cFiles, 'Unexpected number of files');
			AssertEquals(szExpected, lsd.szTotalSize, 'Unexpected file size total');
			mxT := 40;
		ELSE
			TEST_FINISHED();
	END_CASE
END_IF
END_METHOD

METHOD T999_CleanUp
VAR_INPUT
END_VAR
IF TEST_ORDERED('T999_CleanUp') THEN
	IF CleanUp() THEN
		AssertTrue(TRUE, 'cleaned up');
		TEST_FINISHED();
	END_IF
END_IF
END_METHOD

END_FUNCTION_BLOCK

// Device/Application/Mocks/Mock_SyslogRotatingFileHandler
FUNCTION_BLOCK Mock_SyslogRotatingFileHandler EXTENDS Syslog.SyslogRotatingFileHandler
VAR_INPUT
END_VAR
VAR_OUTPUT
END_VAR
VAR
END_VAR

METHOD FileSetup : BOOL
VAR_INPUT
END_VAR
FileSetup := prvFileSetup();
END_METHOD

{attribute 'monitoring' := 'call'}
PROPERTY p_FileSize : UDINT
GET
p_FileSize := THIS^.szFilesize;
END_GET
SET
THIS^.szFilesize := p_FileSize;
END_SET
END_PROPERTY

{attribute 'monitoring' := 'call'}
PROPERTY p_FullFilename : CAA.FILENAME
GET
p_FullFilename := THIS^.sFullFilename;
END_GET
END_PROPERTY

PROPERTY p_hActiveHandle : CAA.HANDLE
GET
p_hActiveHandle := THIS^.hActiveFile;
END_GET
END_PROPERTY

PROPERTY p_mxHandler : UINT
GET
p_mxHandler := mxHandler;
END_GET
END_PROPERTY

PROPERTY p_QueueBusy : BOOL
GET
p_QueueBusy := xQueueBusy;
END_GET
END_PROPERTY

METHOD ProcessQueue : BOOL
VAR_INPUT
END_VAR
ProcessQueue := prvProcessQueue();
END_METHOD

METHOD PubDoRollover : BOOL
VAR_INPUT
END_VAR
PubDoRollover := THIS^.DoRollover();
END_METHOD

METHOD PubRotate : BOOL
VAR_INPUT
	(* The source filename. This is normally the base filename, eg ``test.log``*)
	source	: STRING(255);
	(* The destination filename. This is normally what the source is rotated to, eg ``test.log.1``*)
	dest	: STRING(255);
END_VAR
PubRotate := THIS^.Rotate(source, dest);
END_METHOD

METHOD PubShouldRollover : BOOL
VAR_INPUT
END_VAR
PubShouldRollover := THIS^.ShouldRollover();
END_METHOD

METHOD QueueEmpty : BOOL
VAR_INPUT
END_VAR
QueueEmpty := THIS^.queue.CountElements() = 0;
END_METHOD

METHOD ResetQueue : BOOL
VAR_INPUT
END_VAR
this^.queue.RemoveAllElements();
END_METHOD

END_FUNCTION_BLOCK

// Device/Application/Functions/UT_RandomEmpherialPort
FUNCTION_BLOCK UT_RandomEmpherialPort EXTENDS coUnit.FB_TestSuite
VAR_INPUT
END_VAR
VAR_OUTPUT
END_VAR
VAR
END_VAR

T001_Generate();

METHOD T001_Generate : UINT
VAR_INPUT
END_VAR
VAR_INST
	ix : UINT;
	SortedListFactory : COL.SortedListFactory;
	itfList : COL.ISortedList2;
	UIntElementFactory : COL.UintElementFactory;
	uiResult : UINT;
	iterator : COL.ListIterator;
	itfElem : COL.IElement;
	itfUInt : COL.IUintElement;
	aResult : ARRAY [0..99] OF UINT;
	asResult : ARRAY [0..99] OF UINT;
	xDupSequentialCall : BOOL;
	uiDupSeq : UINT;
	xDup : BOOL;
	uiDup : UINT;
	mxT : UINT;
END_VAR
TEST('T001_Generate');

CASE mxT OF
	0: // init
		IF itfList = 0 THEN
			itfList := SortedListFactory.Create(udiMaxElements:=100);
		END_IF
		mxT := mxT + 10;
	10:
		uiResult := Syslog.RandomEmpherialPort(uiResult);
		aResult[ix] := uiResult;
		itfList.AddElementWithoutSorting(itfElement:=UIntElementFactory.Create(uiValue:=uiResult));
		AssertTrue(uiResult >= 49152 AND uiResult <= 65535, 'Invalid port generated');
		IF ix < 99 THEN
			ix := ix + 1;
		ELSE
			mxT := mxT + 10;
		END_IF
	20:
		itfList.ElementIterator(iterator);
		
		uiResult := 0;
		// Loop through the unsorted list check for duplicates as called
		WHILE iterator.HasNext() DO
			iterator.Next(itfElement=>itfElem);
			__QUERYINTERFACE(itfElem, itfUInt);
			IF uiResult = itfUInt.UintValue THEN
				xDupSequentialCall := TRUE;
				uiDupSeq := uiDupSeq + 1;
			END_IF
			uiResult := itfUInt.UintValue;
		END_WHILE
		
		itfList.Sort();
		itfList.ElementIterator(iterator);
		
		uiResult := 0;
		ix := 0;
		// Loop through the sorted list check for duplicates
		WHILE iterator.HasNext() DO
			iterator.Next(itfElement=>itfElem);
			__QUERYINTERFACE(itfElem, itfUInt);
			IF uiResult = itfUInt.UintValue THEN
				xDup := TRUE;
				uiDup := uiDup + 1;
			END_IF
			uiResult := itfUInt.UintValue;
			asResult[ix] := uiResult;
			ix := ix + 1;
		END_WHILE
		
		AssertFalse(xDup AND xDupSequentialCall, concat('Duplicate port found. How random is this? seq: ', 
													concat(UINT_TO_STRING(uiDupSeq), 
															concat(' dup: ', UINT_TO_STRING(uiDup))))
		);
		mxT := mxT + 10;
	ELSE
		TEST_FINISHED();
END_CASE
END_METHOD

END_FUNCTION_BLOCK

// Device/Application/Function Blocks/UT_SyslogUdpHandler
{attribute 'no_assign'}
FUNCTION_BLOCK UT_SyslogUdpHandler EXTENDS coUnit.FB_TestSuite
VAR_INPUT
END_VAR
VAR_OUTPUT
END_VAR
VAR
	// Adapter IP Address that packets will be sent on
	ipAdapterAddress : NBS.IPv4Address := (ipAddress:='192.168.0.50');
	// Syslog Server IP Address
	ipServerAddress : NBS.IPv4Address := (ipAddress:='192.168.0.10');
	// leave server address out so we can test it missing in T001_Init
	handler : Mock_SyslogUdpHandler := (itfAdapterAddress:=ipAdapterAddress);
END_VAR

T001_Init();
T002_SetupConnection();
T003_ProcessQueue();

METHOD T001_Init
VAR_INPUT
END_VAR
VAR_INST
	mxT : UINT;
END_VAR
IF TEST_ORDERED('T001_Init') THEN
	CASE mxT OF
		0: // Init
			mxT := 10;
		10: // Test with missing Server address
			handler.PubInit();
			mxT := 20;
		20: // Assert error
			AssertTrue(handler.xError, 'Missing server address');
			AssertEquals_STRING('Missing valid adapter or server address', handler.sError, 'Wrong error message');
			handler.Reset();
			handler.itfServerAddress := ipServerAddress;
			mxT := 30;
		30: // check if we can create our async property
			handler.PubInit();
			mxT := 40;
		40: // Expect to get async
			AssertFalse(handler.xError, 'Expected to init without error');
			AssertEquals_STRING('', handler.sError, 'Should have no error message');
			AssertTrue(handler.itfAsyncProperty <> 0, 'Expected valid itfAsyncProperty');
			mxT := 50;
		ELSE
			TEST_FINISHED();
	END_CASE
END_IF
END_METHOD

METHOD T002_SetupConnection
VAR_INPUT
END_VAR
VAR_INST
	mxT : UINT;
	p2Msg : STRING(255);
	eAdSend : NBS.ERROR;
END_VAR
IF TEST_ORDERED('T002_SetupConnection') THEN
	CASE mxT OF 
		0: // Init
			handler.p_uiSendPort := 0;
			handler.PubSetupConnection();
			mxT := 10;
		10: // we should be setup with a random port
			AssertFalse(handler.xError, 'should not have any errors');
			AssertTrue(handler.p_uiSendPort >= 49152 AND handler.p_uiSendPort <= 65535, 'Invalid port generated');
			mxT := 20;
		ELSE
			TEST_FINISHED();
	END_CASE
END_IF
END_METHOD

METHOD T003_ProcessQueue
VAR_INPUT
END_VAR
VAR_INST
	mxT : UINT;
	ix : UINT;
	tmr : TON := (PT:=T#5s);
END_VAR
IF TEST_ORDERED('T003_ProcessQueue') THEN
	CASE mxT OF
		0: // setup
			handler.Dispatch('hello, world');
			handler.Dispatch('<167>1 2021-11-22T23:40:05.003Z codesyslog.example.com UnitTest PLC_PRG DEBUG lorum ipsum');
			mxT := 10;
		10: // run queue process for 5 seconds
			tmr(IN:=TRUE);
			handler.PubProcessQueue();
			IF tmr.Q OR NOT handler.p_QueueBusy THEN
				AssertFalse(tmr.Q, 'ProcessQueue timeout');
				tmr(IN:=FALSE);
				mxT := 20;
			END_IF
		20: // No errors
			AssertFalse(handler.xError, 'Error during queue processing');
			mxT := 30;
		ELSE
			TEST_FINISHED();
	END_CASE
END_IF
END_METHOD

END_FUNCTION_BLOCK

// Device/Application/Mocks/Mock_SyslogUdpHandler
FUNCTION_BLOCK Mock_SyslogUdpHandler EXTENDS Syslog.SyslogUdpHandler
VAR_INPUT
END_VAR
VAR_OUTPUT
END_VAR
VAR
END_VAR

METHOD AdhockSend : NBS.ERROR
VAR_INPUT
	msg : STRING(255);
END_VAR
AdhockSend := THIS^.peer.Send(itfIPAddress:=itfServerAddress, uiPort:=uiPort, pData:=ADR(msg), INT_TO_UDINT(len(msg)));
END_METHOD

PROPERTY p_QueueBusy : BOOL
GET
p_QueueBusy := xQueueBusy;
END_GET
END_PROPERTY

PROPERTY p_uiSendPort : UINT
GET
p_uiSendPort := uiSendPort;
END_GET
SET
uiSendPort := p_uiSendPort;
END_SET
END_PROPERTY

METHOD PUBLIC PubInit : BOOL
VAR_INPUT
END_VAR
PubInit := prvInit();
END_METHOD

METHOD PUBLIC PubProcessQueue : BOOL
VAR_INPUT
END_VAR
PubProcessQueue := prvProcessQueue();
END_METHOD

METHOD PUBLIC PubSetupConnection : BOOL
VAR_INPUT
END_VAR
PubSetupConnection := prvSetupConnection();
END_METHOD

METHOD Reset : BOOL
VAR_INPUT
END_VAR
xError := FALSE;
sError := '';
END_METHOD

END_FUNCTION_BLOCK

// Device/Application/Functions/UT_Make_SdParam
FUNCTION_BLOCK UT_Make_SdParam EXTENDS coUnit.FB_TestSuite
VAR_INPUT
END_VAR
VAR_OUTPUT
END_VAR
VAR
END_VAR

T001_Parameterize('T001_Parameterize:valid', 'varName', 'the value', 'varName="the value"');
T001_Parameterize('T001_Parameterize:escape value', 'varName', '"the value"', 'varName="\"the value\""');
T001_Parameterize('T001_Parameterize:Sanitize_SdName', 'varName ', 'the value', 'varName="the value"');

METHOD T001_Parameterize
VAR_INPUT
	sTestName : STRING(255);
	name : SyslogItfs.PARAM_NAME;
	sValue : STRING(255);
	sExpected : SyslogItfs.STRUCTURED_DATA;
END_VAR

VAR
	sResult : SyslogItfs.STRUCTURED_DATA;
END_VAR
TEST(sTestName);

sResult := Syslog.Make_SdParam(name, ADR(sValue), SIZEOF(sValue));

AssertEquals_STRING(sExpected, sResult, 'unexpected SdParam');

TEST_FINISHED();
END_METHOD

END_FUNCTION_BLOCK

// Device/Application/Functions/UT_Make_SdParam2
FUNCTION_BLOCK UT_Make_SdParam2 EXTENDS coUnit.FB_TestSuite
VAR_INPUT
END_VAR
VAR_OUTPUT
END_VAR
VAR
END_VAR

T001_Parameterize('T001_Parameterize:valid', 'varName', 'the value', 'varName="the value"');
T001_Parameterize('T001_Parameterize:escape value', 'varName', '"the value"', 'varName="\"the value\""');
T001_Parameterize('T001_Parameterize:Sanitize_SdName', 'varName ', 'the value', 'varName="the value"');

METHOD T001_Parameterize
VAR_INPUT
	sTestName : STRING(255);
	name : SyslogItfs.PARAM_NAME;
	sValue : STRING(255);
	sExpected : SyslogItfs.STRUCTURED_DATA;
END_VAR

VAR
	sResult : SyslogItfs.STRUCTURED_DATA;
END_VAR
TEST(sTestName);

sResult := Syslog.Make_SdParam2(name, sValue);

AssertEquals_STRING(sExpected, sResult, 'unexpected SdParam2');

TEST_FINISHED();
END_METHOD

END_FUNCTION_BLOCK

// Device/Application/Functions/UT_StrucDataMsg
FUNCTION_BLOCK UT_StrucDataMsg EXTENDS coUnit.FB_TestSuite
VAR_INPUT
END_VAR
VAR_OUTPUT
END_VAR
VAR

END_VAR

T001_Parameterize('T001_Parameterize:full_length', uiMsgLength:=SyslogItfs.gc_szMsg-1024, uiMsgTruncLength:=SyslogItfs.gc_szMsg-1024);
T001_Parameterize('T001_Parameterize:trunc_length', uiMsgLength:=1024, uiMsgTruncLength:=SyslogItfs.gc_szMsg-1024);
T001_Parameterize('T001_Parameterize:short_length', uiMsgLength:=255, uiMsgTruncLength:=255);

METHOD AssertEquals_SyslogMsg
VAR_INPUT
	actual : POINTER TO SyslogItfs.SYSLOG_MSG;
	expected : POINTER TO SyslogItfs.SYSLOG_MSG;
END_VAR
VAR
	ix : UINT;
	pa : POINTER TO ARRAY [0..SyslogItfs.gc_szSyslogMsg-1] OF BYTE := actual;
	pe : POINTER TO ARRAY [0..SyslogItfs.gc_szSyslogMsg-1] OF BYTE := expected;
	xDifferent : BOOL;
END_VAR
FOR ix := 0 TO SyslogItfs.gc_szSyslogMsg-1 BY 1 DO
	IF pa^[ix] <> 0 AND pe^[ix] <> 0 THEN
		IF pa^[ix] <> pe^[ix] THEN
			xDifferent := TRUE;
			EXIT;
		END_IF
	ELSIF pa^[ix] = 0 AND pe^[ix] = 0 THEN
		EXIT;
	ELSE
		xDifferent := TRUE;
		EXIT;
	END_IF
END_FOR

AssertFalse(xDifferent, concat('SYSLOG_MSG found to differ at character: ', UINT_TO_STRING(ix)));
END_METHOD

METHOD T001_Parameterize
VAR_INPUT
	sTestName : STRING(255);
	uiMsgLength : UINT;
	uiMsgTruncLength : UINT;
END_VAR

VAR
	sd : Mock_StructuredData := (uiMsgLength:=1024);
	msgMaker : Mock_MsgPrependSpace := (fill:=121);
	msg : SyslogItfs.MSG;
	sExpected : SyslogItfs.MSG;
	sResult : SyslogItfs.MSG;
END_VAR
TEST(sTestName);

// Make expected result
sExpected := sd.AsStructuredData();
msgMaker.uiMsgLength := MIN(SyslogItfs.gc_szMsg, uiMsgTruncLength);
msg := msgMaker.AsStructuredData();
Stu.StrConcatA(pstFrom:=ADR(msg), pstTo:=ADR(sExpected), SIZEOF(sExpected));
// Actual msg length
msgMaker.uiMsgLength := MIN(SyslogItfs.gc_szMsg, uiMsgLength);
msg := msgMaker.AsStructuredData();
Stu.StrTrimStartA(ADR(msg));

// run the function
sResult := Syslog.StrucDataMsg(sd, msg);

AssertEquals_SyslogMsg(ADR(sResult), ADR(sExpected));

TEST_FINISHED();
END_METHOD

END_FUNCTION_BLOCK

// Device/Application/Mocks/Mock_StructuredData
FUNCTION_BLOCK Mock_StructuredData IMPLEMENTS SyslogItfs.IStructuredData
VAR_INPUT
	uiMsgLength : UINT;
	fill : BYTE := 120;
END_VAR
VAR_OUTPUT
END_VAR
VAR
END_VAR

(* Create a RFC5424 Structured Data Element*)
METHOD AsStructuredData : SyslogItfs.STRUCTURED_DATA
VAR
	pby : POINTER TO ARRAY [0..SyslogItfs.gc_szStructuredData] OF BYTE;
	ix : UINT;
END_VAR
AsStructuredData := 'x';
pby := ADR(AsStructuredData);
FOR ix := 0 TO MIN(uiMsgLength-1, (SyslogItfs.gc_szStructuredData-1)) BY 1 DO
	pby^[ix] := fill;
END_FOR
// null terminate
pby^[ix] := 0;
END_METHOD

END_FUNCTION_BLOCK

// Device/Application/Mocks/Mock_MsgPrependSpace
FUNCTION_BLOCK Mock_MsgPrependSpace IMPLEMENTS SyslogItfs.IStructuredData
VAR_INPUT
	uiMsgLength : UINT;
	fill : BYTE := 120;
END_VAR
VAR_OUTPUT
END_VAR
VAR
END_VAR

(* Create a RFC5424 Structured Data Element*)
METHOD AsStructuredData : SyslogItfs.STRUCTURED_DATA
VAR
	pby : POINTER TO ARRAY [0..SyslogItfs.gc_szStructuredData] OF BYTE;
	ix : UINT;
END_VAR
AsStructuredData := ' ';
pby := ADR(AsStructuredData);
FOR ix := 1 TO MIN(uiMsgLength-1, (SyslogItfs.gc_szStructuredData-1)) BY 1 DO
	pby^[ix] := fill;
END_FOR
// null terminate
pby^[ix] := 0;
END_METHOD

END_FUNCTION_BLOCK

// Device/Application/Function Blocks/UT_SyslogAlarmOnMessageHandler
FUNCTION_BLOCK UT_SyslogAlarmOnMessageHandler EXTENDS coUnit.FB_TestSuite
VAR_INPUT
END_VAR
VAR_OUTPUT
END_VAR
VAR
	handler : SyslogAlarmOnMessage.SyslogAlarmOnMessageHandler := (severity:=SyslogItfs.SyslogSeverity.DEBUG);
	logger : Syslog.SyslogLogger(hostname:='unittest', appName:='AlarmOn', procId:='-', facility:=SyslogItfs.SyslogFacility.LOCAL1, handler:=handler);
	xtTrip : PceAlarms.TripAlarm;
	xwWarn : PceAlarms.WarnAlarm;
	xeError : PceAlarms.RepeatToAlarm := (iMaxError:=10);
	xInit : BOOL;
END_VAR

IF NOT xInit THEN
	handler.Register(xtTrip, 'TRIP');
	handler.Register(xwWarn, 'WARN');
	handler.Register(xeError, 'REPEAT');
	xInit := TRUE;
END_IF

T001_TripAlarm();
T002_WarnAlarm();
T003_RepeatAlarm();
T004_RegisterDup();

METHOD T001_TripAlarm
VAR_INPUT
END_VAR
TEST('T001_TripAlarm');

logger.Error('TripAlarm', 'TRIP on this message');
xtTrip();
AssertTrue(xtTrip.p_xTrip, 'Should be tripped');

xtTrip.xError := FALSE;
xtTrip.Reset();
logger.Warning('TripAlarm', 'no trip here');
xtTrip();
AssertFalse(xtTrip.p_xTrip, 'Should NOT be tripped');
AssertFalse(xwWarn.p_xWarn, 'xwWarn should not be set');
AssertEquals_INT(0, xeError.iErrorCount, 'xeError should not have any count');

TEST_FINISHED();
END_METHOD

METHOD T002_WarnAlarm
VAR_INPUT
END_VAR
TEST('T002_WarnAlarm');

logger.Error('T002_WarnAlarm', 'WARN on this message');
xwWarn();
AssertTrue(xwWarn.p_xWarn, 'Should be warning');

xwWarn.xError := FALSE;
xwWarn.Reset();
logger.Warning('T002_WarnAlarm', 'no warn here');
xtTrip();
xwWarn();
xeError();
AssertFalse(xtTrip.p_xTrip, 'Should NOT be tripped');
AssertFalse(xwWarn.p_xWarn, 'xwWarn should not be set');
AssertEquals_INT(0, xeError.iErrorCount, 'xeError should not have any count');

TEST_FINISHED();
END_METHOD

METHOD T003_RepeatAlarm
VAR_INPUT
END_VAR
VAR
	ix : INT;
END_VAR
TEST('T003_RepeatAlarm');

FOR ix:=1 TO 9 BY 1 DO
	logger.Error('T003_RepeatAlarm', PSB.Format_1('REPEAT on this message: {}', TO_STRING(ix)));
	AssertEquals_INT(ix, xeError.iErrorCount, 'Unexpected xeError.iErrorCount');
	AssertTrue(xeError.p_xWarn, PSB.Format_1('Should be in warn {}', TO_STRING(ix)));
	AssertFalse(xeError.p_xTrip, PSB.Format_1('Should not be in trip {}', TO_STRING(ix)));
END_FOR

ix := 10;
logger.Error('T003_RepeatAlarm', PSB.Format_1('REPEAT on this message: {}', TO_STRING(ix)));
AssertEquals_INT(ix, xeError.iErrorCount, 'Unexpected xeError.iErrorCount');
AssertTrue(xeError.p_xWarn, PSB.Format_1('Should be in warn {}', TO_STRING(ix)));
AssertTrue(xeError.p_xTrip, PSB.Format_1('Should not be in trip {}', TO_STRING(ix)));

xtTrip();
xwWarn();
AssertFalse(xtTrip.p_xTrip, 'Should NOT be tripped');
AssertFalse(xwWarn.p_xWarn, 'xwWarn should not be set');


TEST_FINISHED();
END_METHOD

METHOD T004_RegisterDup
VAR_INPUT
END_VAR
TEST('T004_RegisterDup');

AssertEquals_INT(ENO.errno.EALREADY, handler.Register(xeError, 'REPEAT'), 'Unexpected return from handler.Register');

TEST_FINISHED();
END_METHOD

END_FUNCTION_BLOCK

// Device/Application/Function Blocks/UT_SyslogCaaUdpHandler
{attribute 'no_assign'}
FUNCTION_BLOCK UT_SyslogCaaUdpHandler EXTENDS coUnit.FB_TestSuite
VAR_INPUT
END_VAR
VAR_OUTPUT
END_VAR
VAR
	// leave server address out so we can test it missing in T001_Init
	handler : Mock_SyslogCaaUdpHandler := (sIpAddress:='192.168.0.10');
END_VAR

T002_SetupConnection();
T003_ProcessQueue();

METHOD T002_SetupConnection
VAR_INPUT
END_VAR
VAR_INST
	mxT : UINT;
	p2Msg : STRING(255);
	eAdSend : NBS.ERROR;
END_VAR
IF TEST_ORDERED('T002_SetupConnection') THEN
	CASE mxT OF 
		0: // Init
			handler.p_uiSendPort := 0;
			handler.PubSetupConnection();
			mxT := 10;
		10: // we should be setup with a random port
			AssertFalse(handler.xError, 'should not have any errors');
			AssertTrue(handler.p_uiSendPort >= 49152 AND handler.p_uiSendPort <= 65535, 'Invalid port generated');
			mxT := 20;
		ELSE
			TEST_FINISHED();
	END_CASE
END_IF
END_METHOD

METHOD T003_ProcessQueue
VAR_INPUT
END_VAR
VAR_INST
	mxT : UINT;
	ix : UINT;
	tmr : TON := (PT:=T#5s);
END_VAR
IF TEST_ORDERED('T003_ProcessQueue') THEN
	CASE mxT OF
		0: // setup
			handler.Dispatch('hello, world CAA');
			handler.Dispatch('<167>1 2021-11-22T23:40:05.003Z codesyslog.example.com UnitTest PLC_PRG DEBUG lorum ipsum CAA');
			mxT := 10;
		10: // run queue process for 5 seconds
			tmr(IN:=TRUE);
			handler.PubProcessQueue();
			IF tmr.Q OR NOT handler.p_QueueBusy THEN
				AssertFalse(tmr.Q, 'ProcessQueue timeout');
				tmr(IN:=FALSE);
				mxT := 20;
			END_IF
		20: // No errors
			AssertFalse(handler.xError, 'Error during queue processing');
			mxT := 30;
		ELSE
			TEST_FINISHED();
	END_CASE
END_IF
END_METHOD

END_FUNCTION_BLOCK

// Device/Application/Mocks/Mock_SyslogCaaUdpHandler
FUNCTION_BLOCK Mock_SyslogCaaUdpHandler EXTENDS SyslogCaaHandlers.SyslogCaaUdpHandler
VAR_INPUT
END_VAR
VAR_OUTPUT
END_VAR
VAR
END_VAR

PROPERTY p_QueueBusy : BOOL
GET
p_QueueBusy := xQueueBusy;
END_GET
END_PROPERTY

PROPERTY p_uiSendPort : UINT
GET
p_uiSendPort := uiSendPort;
END_GET
SET
uiSendPort := p_uiSendPort;
END_SET
END_PROPERTY

METHOD PUBLIC PubProcessQueue : BOOL
VAR_INPUT
END_VAR
PubProcessQueue := prvProcessQueue();
END_METHOD

METHOD PUBLIC PubSetupConnection : BOOL
VAR_INPUT
END_VAR
PubSetupConnection := prvSetupConnection();
END_METHOD

METHOD Reset : BOOL
VAR_INPUT
END_VAR
xError := FALSE;
sError := '';
END_METHOD

END_FUNCTION_BLOCK
